FUNCTION_BLOCK TestMotion
VAR_IN_OUT
	axis  : ARRAY [XP .. XM] OF AxisGroup;
	nextInstruct, abortRequest, resetRequest, startRequest, stopRequest: BOOL;
	homeRequest : BYTE;
		
	//statemachine
	stateLVL1 : INT;
	
END_VAR
VAR_INPUT

	speed : LREAL;	

END_VAR
VAR_OUTPUT
END_VAR
VAR
	 //used in tracking Action
	 xorResult : BOOL;
	
	//state-machine
	stateLVL2 : INT;
	initStateLVL2 : BOOL;
	motionBusy : BOOL;
	
	//counter
	i 	: INT :=0;
	
	//used in homeShutter Action
	homeDelay : TON;

END_VAR
VAR CONSTANT
	BRAKE_OFF_C		: BOOL	:= TRUE;
	BRAKE_ON_C		: BOOL	:= FALSE;
	SCAN_VEL_C		: LREAL := 60;
	HOME_VEL_C		: LREAL	:= 3;
	CALIBRATE_VEL_C	: LREAL	:= 100;
	POSITION_VEL_C	: LREAL := 300;
	POS_START_C		: LREAL := 0;
	POS_END_C		: LREAL := 751;
	HOMEOFFSET_XP_C	: LREAL	:= (POS_START_C+35);
	HOMEOFFSET_XM_C	: LREAL	:= (POS_END_C-84);
	
	//SIZE_HALL_SW_C 	: LREAL := SIZEOF(GVL.hallPosCalXP);
	
	//For indexing axis
	XP : INT := 0;
	XM : INT := 1;
END_VAR

(*
This function block contains all the motion of the shutter. There are two state machine in this module - stateLVL1 and stateLVL2.
stateLVL1 is used to switch between motions. stateLVL2 is used to operate the statemachine within the particular motion.
Motions are split into different action objects for readibility and maintainability. 
*)

//update Axis_Ref status
axis[XP].axisRef.ReadStatus();
axis[XM].axisRef.ReadStatus();

//reset input
IF abortRequest THEN
	abortRequest := FALSE;
	stateLVL1 := -1; 
END_IF
IF resetRequest THEN
	resetRequest := FALSE;
	stateLVL1 := 0;
END_IF

(*Case statement for motions. There are two level of state. LVL1 located here and LVL2 which are in the ACTION files.*)
CASE stateLVL1 OF
	-1: //Abort state. Disable movement
		axis[XP].mcPower(Axis := axis[XP].axisRef, Enable := TRUE, Enable_Positive := FALSE, Enable_Negative := FALSE);
		axis[XM].mcPower(Axis := axis[XM].axisRef, Enable := TRUE, Enable_Positive := FALSE, Enable_Negative := FALSE);	
		axis[XP].mcHome(Axis := axis[XP].axisRef, Execute := FALSE);
		axis[XM].mcHome(Axis := axis[XP].axisRef, Execute := FALSE);
		axis[XP].mcReset(Axis := axis[XP].axisRef, Execute := FALSE);
		axis[XM].mcReset(Axis := axis[XM].axisRef, Execute := FALSE);
		axis[XP].brake 	:= BRAKE_ON_C;
		axis[XM].brake 	:= BRAKE_ON_C;
		nextInstruct 	:= FALSE;
		GVL.fbWaitTimer(IN:=FALSE);
		
	0: //reset state
		motionBusy := FALSE;
		initStateLVL2 := FALSE;
		nextInstruct := FALSE;
		axis[XP].mcReset(Axis := axis[XP].axisRef, Execute := TRUE, ErrorID => axis[XP].errorID);
		axis[XM].mcReset(Axis := axis[XM].axisRef, Execute := TRUE, ErrorID => axis[XM].errorID);
		IF axis[XP].mcReset.Error OR axis[XM].mcReset.Error THEN
			axis[XP].mcPower(Axis := axis[XP].axisRef, Enable := TRUE, Enable_Positive := FALSE, Enable_Negative := FALSE);
			axis[XM].mcPower(Axis := axis[XM].axisRef, Enable := TRUE, Enable_Positive := FALSE, Enable_Negative := FALSE);
			axis[XP].brake 	:= BRAKE_ON_C;
			axis[XM].brake 	:= BRAKE_ON_C;
			stateLVL1 		:= -1; //go to stop state
			stateLVL2		:=0;

			//Should report an error flag go to error handle state
		ELSIF axis[XP].mcReset.Done AND axis[XM].mcReset.Done THEN
			axis[XP].mcPower(Axis := axis[XP].axisRef, Enable := TRUE, Enable_Positive := TRUE, Enable_Negative := TRUE);
			axis[XM].mcPower(Axis := axis[XM].axisRef, Enable := TRUE, Enable_Positive := TRUE, Enable_Negative := TRUE);
			axis[XP].mcReset(Axis := axis[XP].axisRef, Execute := FALSE);
			axis[XM].mcReset(Axis := axis[XM].axisRef, Execute := FALSE);
			axis[XP].brake := BRAKE_OFF_C;
			axis[XM].brake := BRAKE_OFF_C;
			axis[XP].mcStop(Axis:=axis[XP].axisRef, Execute:=FALSE);
			axis[XM].mcStop(Axis:=axis[XM].axisRef, Execute:=FALSE);
			stateLVL1 	:= 100; //go to stop state
			stateLVL2	:=0;		
			GVL.fbWaitTimer(IN:=FALSE);	
		END_IF
		
	100: //stop state
		axis[XP].mcMoveAbs(Axis := axis[XP].axisRef, Execute := FALSE);
		axis[XM].mcMoveAbs(Axis := axis[XM].axisRef, Execute := FALSE);
		axis[XP].mcJog(Axis:=axis[XP].axisRef, JogForward:=FALSE, JogBackwards:=FALSE);
		axis[XM].mcJog(Axis:=axis[XM].axisRef, JogForward:=FALSE, JogBackwards:=FALSE);
		axis[XP].mcHome(Axis := axis[XP].axisRef, Execute := FALSE);
		axis[XM].mcHome(Axis := axis[XP].axisRef, Execute := FALSE);
		stateLVL2 := 0;
		GVL.fbWaitTimer(IN:=FALSE);
	
	400: //Homing start for both blades
		homeShutter();
		IF motionBusy = FALSE THEN
			stateLVL1:=100;
		END_IF


	//States higher than 400 requires HOMING ROUTINE to be ran first.
	//////////////////////////////////////////////////////////////////////////////////////////////
	//Basic Motions
	//////////////////////////////////////////////////////////////////////////////////////////////	

	1000: //Open shutter
		openShutter();
		IF motionBusy = FALSE THEN
			stateLVL1:=100;
		END_IF
		
	1100: //Close shutter towards X+ side. 
		closeShutterPlus();
		IF motionBusy = FALSE THEN
			stateLVL1:=100;
		END_IF
		
	1200: //Close shutter towards X- side. 
		closeShutterMinus();
		IF motionBusy = FALSE THEN
			stateLVL1:=100;
		END_IF
		
	1300: //AxisXP absolute move
		axis[XP].mcMoveAbs(Axis:=axis[XP].axisRef, Position:=GVL.setPosition, Velocity:=speed, Execute:=TRUE);
		IF axis[XP].mcMoveAbs.Done THEN
			axis[XP].mcMoveAbs(Axis:=axis[XP].axisRef, Execute:=FALSE);
			stateLVL1 := 100;
		END_IF

	1400: //AxisXM move absolute
		axis[XM].mcMoveAbs(Axis:=axis[XM].axisRef, Position:=GVL.setPosition, Velocity:=speed, Execute:=TRUE);
		IF axis[XM].mcMoveAbs.Done THEN
			axis[XM].mcMoveAbs(Axis:=axis[XM].axisRef, Execute:=FALSE);
			stateLVL1 := 100;
		END_IF

	1500: //AxisXP Jog Forward
		axis[XP].mcJog(Axis:=axis[XP].axisRef, JogForward:=TRUE, JogBackwards:=FALSE, Mode:=MC_JOGMODE_STANDARD_SLOW);
	
	1600: //AxisXP Jog Backward
		axis[XP].mcJog(Axis:=axis[XP].axisRef, JogForward:=FALSE, JogBackwards:=TRUE, Mode:=MC_JOGMODE_STANDARD_SLOW);
		
	1700: //AxisXM Jog Backward
		axis[XM].mcJog(Axis:=axis[XM].axisRef, JogForward:=TRUE, JogBackwards:=FALSE, Mode:=MC_JOGMODE_STANDARD_SLOW);
	
	1800: //AxisXM Jog Forward
		axis[XM].mcJog(Axis:=axis[XM].axisRef, JogForward:=FALSE, JogBackwards:=TRUE, Mode:=MC_JOGMODE_STANDARD_SLOW);

	
	//////////////////////////////////////////////////////////////////////////////////////////////
	//Motion for visit - NORMAL MODE
	//////////////////////////////////////////////////////////////////////////////////////////////	

	2000:
		visit();
		IF motionBusy = FALSE THEN
			stateLVL1:=100;
		END_IF
	
	//////////////////////////////////////////////////////////////////////////////////////////////
	//Cycler -- for use in testing shutter cycle
	//////////////////////////////////////////////////////////////////////////////////////////////
		
	3100: //Cycler sequence 
		cycler();
		IF motionBusy = FALSE THEN
			stateLVL1:=100;
		END_IF	

	//////////////////////////////////////////////////////////////////////////////////////////////
	//Soft Calibration
	//////////////////////////////////////////////////////////////////////////////////////////////

	8000: //Perform soft calibration
		calibrateXP();
		calibrateXM();
		//openShutter();
		IF motionBusy = FALSE THEN
			stateLVL1:=100;
		END_IF

END_CASE

//track motion of both blades
tracking();

ACTION calibrateXM:
//////////////////////////////////////////////////
//perform software calibration of axisXM blade. //
//////////////////////////////////////////////////

IF initStateLVL2 = FALSE THEN
	initStateLVL2 := TRUE;
	stateLVL2 :=9010;
	motionBusy := TRUE;
END_IF	

CASE stateLVL2 OF
	
	9010: //Clear previous Calibration value
		FOR i:=0 TO GVL.tripCount_C BY 1 DO
			axis[XM].hallPosCal[0,i]:=0;
			axis[XM].hallPosCal[1,i]:=0;
		END_FOR
		axis[XM].tripCount := 0;
		axis[XM].isCalibrated := FALSE;
		stateLVL2:=9020;
		
	9020: //Put Shutter in Open Position
		axis[XP].mcMoveAbs(Axis:=axis[XP].axisRef, Position:= POS_START_C, Velocity:=POSITION_VEL_C, Execute:=TRUE);
		axis[XM].mcMoveAbs(Axis:=axis[XM].axisRef, Position:= POS_END_C, Velocity:=POSITION_VEL_C, Execute:=TRUE);
		IF axis[XP].mcMoveAbs.Done AND axis[XM].mcMoveAbs.Done THEN
			axis[XP].mcMoveAbs(Axis:=axis[XP].axisRef, Execute:=FALSE);
			axis[XM].mcMoveAbs(Axis:=axis[XM].axisRef, Execute:=FALSE);
			stateLVL2:=9030;
		END_IF
		
		//This section is required to get rid of false trigger when system starts up
		FOR i:=GVL.hallLower_C TO GVL.hallUpper_C BY 1 DO
			axis[XM].hallSigCal_rtrig[i](CLK:=GVL.hallSwitch[i]);
			axis[XM].hallSigCal_ftrig[i](CLK:=GVL.hallSwitch[i]);
			IF axis[XM].hallSigCal_rtrig[i].Q OR axis[XM].hallSigCal_ftrig[i].Q THEN
				; //do nothing
			END_IF
		END_FOR	
	
	9030: //Calibrate AxisXM twoards X+ side.
		//record position and sequence of hall trips at rising and falling edge.
		FOR i:=GVL.hallLower_C TO GVL.hallUpper_C BY 1 DO
			axis[XM].hallSigCal_rtrig[i](CLK:=GVL.hallSwitch[i]);
			axis[XM].hallSigCal_ftrig[i](CLK:=GVL.hallSwitch[i]);
			IF axis[XM].hallSigCal_rtrig[i].Q OR axis[XM].hallSigCal_ftrig[i].Q THEN	
				
				axis[XM].hallSequence[GVL.dirNeg_C, axis[XM].tripCount].0 := axis[XM].hallSigCal_rtrig[0].Q OR axis[XM].hallSigCal_ftrig[0].Q;
				axis[XM].hallSequence[GVL.dirNeg_C, axis[XM].tripCount].1 := axis[XM].hallSigCal_rtrig[1].Q OR axis[XM].hallSigCal_ftrig[1].Q;
				axis[XM].hallSequence[GVL.dirNeg_C, axis[XM].tripCount].2 := axis[XM].hallSigCal_rtrig[2].Q OR axis[XM].hallSigCal_ftrig[2].Q;
				axis[XM].hallSequence[GVL.dirNeg_C, axis[XM].tripCount].3 := axis[XM].hallSigCal_rtrig[3].Q OR axis[XM].hallSigCal_ftrig[3].Q;
				axis[XM].hallSequence[GVL.dirNeg_C, axis[XM].tripCount].4 := axis[XM].hallSigCal_rtrig[4].Q OR axis[XM].hallSigCal_ftrig[4].Q;
				axis[XM].hallSequence[GVL.dirNeg_C, axis[XM].tripCount].5 := axis[XM].hallSigCal_rtrig[5].Q OR axis[XM].hallSigCal_ftrig[5].Q;
				axis[XM].hallSequence[GVL.dirNeg_C, axis[XM].tripCount].6 := axis[XM].hallSigCal_rtrig[6].Q OR axis[XM].hallSigCal_ftrig[6].Q;
				axis[XM].hallSequence[GVL.dirNeg_C, axis[XM].tripCount].7 := axis[XM].hallSigCal_rtrig[7].Q OR axis[XM].hallSigCal_ftrig[7].Q;
				axis[XM].hallSequence[GVL.dirNeg_C, axis[XM].tripCount].8 := axis[XM].hallSigCal_rtrig[8].Q OR axis[XM].hallSigCal_ftrig[8].Q;
				axis[XM].hallSequence[GVL.dirNeg_C, axis[XM].tripCount].9 := axis[XM].hallSigCal_rtrig[9].Q OR axis[XM].hallSigCal_ftrig[9].Q;
				axis[XM].hallSequence[GVL.dirNeg_C, axis[XM].tripCount].10 := axis[XM].hallSigCal_rtrig[10].Q OR axis[XM].hallSigCal_ftrig[10].Q;
				axis[XM].hallSequence[GVL.dirNeg_C, axis[XM].tripCount].11 := axis[XM].hallSigCal_rtrig[11].Q OR axis[XM].hallSigCal_ftrig[11].Q;
				axis[XM].hallSequence[GVL.dirNeg_C, axis[XM].tripCount].12 := axis[XM].hallSigCal_rtrig[12].Q OR axis[XM].hallSigCal_ftrig[12].Q;
				axis[XM].hallSequence[GVL.dirNeg_C, axis[XM].tripCount].13 := axis[XM].hallSigCal_rtrig[13].Q OR axis[XM].hallSigCal_ftrig[13].Q;
				axis[XM].hallSequence[GVL.dirNeg_C, axis[XM].tripCount].14 := axis[XM].hallSigCal_rtrig[14].Q OR axis[XM].hallSigCal_ftrig[14].Q;
				
				axis[XM].hallPosCal[GVL.dirNeg_C, axis[XM].tripCount] := axis[XM].axisRef.NcToPlc.ActPos;
				
				axis[XM].tripCount := axis[XM].tripCount + 1;		

			END_IF
		END_FOR

		//start moving axisXP towards x+ side
		axis[XM].mcMoveAbs(Axis:=axis[XM].axisRef, Position:=POS_START_C, Velocity:=CALIBRATE_VEL_C, Execute:=TRUE);
		IF axis[XM].mcMoveAbs.Done THEN
			axis[XM].mcMoveAbs(Axis:=axis[XP].axisRef, Execute:=FALSE);
			stateLVL2:= 9040;
		END_IF
	
	
	9040: //Calibrate AxisXM twoards X- side.
		//record position and sequence of hall trips at rising and falling edge.
		FOR i:=GVL.hallLower_C TO GVL.hallUpper_C BY 1 DO
			axis[XM].hallSigCal_rtrig[i](CLK:=GVL.hallSwitch[i]);
			axis[XM].hallSigCal_ftrig[i](CLK:=GVL.hallSwitch[i]);
			IF axis[XM].hallSigCal_rtrig[i].Q OR axis[XM].hallSigCal_ftrig[i].Q THEN	
				
				axis[XM].hallSequence[GVL.dirPos_C, axis[XM].tripCount].0 := axis[XM].hallSigCal_rtrig[0].Q OR axis[XM].hallSigCal_ftrig[0].Q;
				axis[XM].hallSequence[GVL.dirPos_C, axis[XM].tripCount].1 := axis[XM].hallSigCal_rtrig[1].Q OR axis[XM].hallSigCal_ftrig[1].Q;
				axis[XM].hallSequence[GVL.dirPos_C, axis[XM].tripCount].2 := axis[XM].hallSigCal_rtrig[2].Q OR axis[XM].hallSigCal_ftrig[2].Q;
				axis[XM].hallSequence[GVL.dirPos_C, axis[XM].tripCount].3 := axis[XM].hallSigCal_rtrig[3].Q OR axis[XM].hallSigCal_ftrig[3].Q;
				axis[XM].hallSequence[GVL.dirPos_C, axis[XM].tripCount].4 := axis[XM].hallSigCal_rtrig[4].Q OR axis[XM].hallSigCal_ftrig[4].Q;
				axis[XM].hallSequence[GVL.dirPos_C, axis[XM].tripCount].5 := axis[XM].hallSigCal_rtrig[5].Q OR axis[XM].hallSigCal_ftrig[5].Q;
				axis[XM].hallSequence[GVL.dirPos_C, axis[XM].tripCount].6 := axis[XM].hallSigCal_rtrig[6].Q OR axis[XM].hallSigCal_ftrig[6].Q;
				axis[XM].hallSequence[GVL.dirPos_C, axis[XM].tripCount].7 := axis[XM].hallSigCal_rtrig[7].Q OR axis[XM].hallSigCal_ftrig[7].Q;
				axis[XM].hallSequence[GVL.dirPos_C, axis[XM].tripCount].8 := axis[XM].hallSigCal_rtrig[8].Q OR axis[XM].hallSigCal_ftrig[8].Q;
				axis[XM].hallSequence[GVL.dirPos_C, axis[XM].tripCount].9 := axis[XM].hallSigCal_rtrig[9].Q OR axis[XM].hallSigCal_ftrig[9].Q;
				axis[XM].hallSequence[GVL.dirPos_C, axis[XM].tripCount].10 := axis[XM].hallSigCal_rtrig[10].Q OR axis[XM].hallSigCal_ftrig[10].Q;
				axis[XM].hallSequence[GVL.dirPos_C, axis[XM].tripCount].11 := axis[XM].hallSigCal_rtrig[11].Q OR axis[XM].hallSigCal_ftrig[11].Q;
				axis[XM].hallSequence[GVL.dirPos_C, axis[XM].tripCount].12 := axis[XM].hallSigCal_rtrig[12].Q OR axis[XM].hallSigCal_ftrig[12].Q;
				axis[XM].hallSequence[GVL.dirPos_C, axis[XM].tripCount].13 := axis[XM].hallSigCal_rtrig[13].Q OR axis[XM].hallSigCal_ftrig[13].Q;
				axis[XM].hallSequence[GVL.dirPos_C, axis[XM].tripCount].14 := axis[XM].hallSigCal_rtrig[14].Q OR axis[XM].hallSigCal_ftrig[14].Q;
			
				axis[XM].hallPosCal[GVL.dirPos_C, axis[XM].tripCount] := axis[XM].axisRef.NcToPlc.ActPos;
				axis[XM].tripCount := axis[XM].tripCount - 1;	
			END_IF
		END_FOR
	
		//start moving axisXP towards x- side
		axis[XM].mcMoveAbs(Axis:=axis[XM].axisRef, Position:=POS_END_C, Velocity:=CALIBRATE_VEL_C, Execute:=TRUE);
		IF axis[XM].mcMoveAbs.Done THEN
			axis[XM].mcMoveAbs(Axis:=axis[XM].axisRef, Execute:=FALSE);
			stateLVL2 := 9050;
		END_IF
		
	9050: 
		axis[XM].mcJog(Axis := axis[XM].axisRef, Mode := MC_JOGMODE_CONTINOUS, Velocity := SCAN_VEL_C, JogBackwards := axis[XM].limitHome);
		IF NOT axis[XM].limitHome THEN
			axis[XM].mcJog(Axis := axis[XM].axisRef, Mode := MC_JOGMODE_CONTINOUS, JogBackwards := FALSE);
			stateLVL2 := 9060;
		END_IF

	9060: //slowly homed back to switch
		axis[XM].mcJog(Axis := axis[XM].axisRef, Mode := MC_JOGMODE_CONTINOUS, Velocity := HOME_VEL_C, JogForward := NOT axis[XM].limitHome);
		IF axis[XM].limitHome THEN
			axis[XM].mcJog(Axis := axis[XM].axisRef, Mode := MC_JOGMODE_CONTINOUS, JogForward := FALSE);
			stateLVL2 := 9070;
			axis[XM].isCalibrated := TRUE;
		END_IF			
		
	9070: //End action
		initStateLVL2 := FALSE;
		stateLVL2 := 0;
		motionBusy := FALSE;


END_CASE
END_ACTION

ACTION calibrateXP:
//////////////////////////////////////////////////
//perform software calibration of axisXP blade. //
//////////////////////////////////////////////////

IF initStateLVL2 = FALSE THEN
	initStateLVL2 := TRUE;
	stateLVL2 :=8010;
	motionBusy := TRUE;
END_IF	

CASE stateLVL2 OF

	8010: //Clear previous Calibration value
		FOR i:=0 TO GVL.tripCount_C BY 1 DO
			axis[XP].hallPosCal[0,i]:=0;
			axis[XP].hallPosCal[1,i]:=0;
		END_FOR
		axis[XP].tripCount := 0;	
		axis[XP].isCalibrated := FALSE;
		stateLVL2:=8020;
		
	8020: //Put Shutter in Open Position
		axis[XP].mcMoveAbs(Axis:=axis[XP].axisRef, Position:= POS_START_C, Velocity:=POSITION_VEL_C, Execute:=TRUE);
		axis[XM].mcMoveAbs(Axis:=axis[XM].axisRef, Position:= POS_END_C, Velocity:=POSITION_VEL_C, Execute:=TRUE);
		IF axis[XP].mcMoveAbs.Done AND axis[XM].mcMoveAbs.Done THEN
			axis[XP].mcMoveAbs(Axis:=axis[XP].axisRef, Execute:=FALSE);
			axis[XM].mcMoveAbs(Axis:=axis[XM].axisRef, Execute:=FALSE);
			stateLVL2:=8030;
		END_IF
		
		//This section is required to get rid of false trigger when system starts up
		FOR i:=GVL.hallLower_C TO GVL.hallUpper_C BY 1 DO
			axis[XP].hallSigCal_rtrig[i](CLK:=GVL.hallSwitch[i]);
			axis[XP].hallSigCal_ftrig[i](CLK:=GVL.hallSwitch[i]);
			IF axis[XP].hallSigCal_rtrig[i].Q OR axis[XP].hallSigCal_ftrig[i].Q THEN
				; //do nothing
			END_IF
		END_FOR

	8030: //Calibrate AxisXP towards X- side.
		//record position and sequence of hall trips at rising and falling edge.
		FOR i:=GVL.hallLower_C TO GVL.hallUpper_C BY 1 DO
			axis[XP].hallSigCal_rtrig[i](CLK:=GVL.hallSwitch[i]);
			axis[XP].hallSigCal_ftrig[i](CLK:=GVL.hallSwitch[i]);
			IF axis[XP].hallSigCal_rtrig[i].Q OR axis[XP].hallSigCal_ftrig[i].Q THEN	

				axis[XP].hallSequence[GVL.dirPos_C, axis[XP].tripCount].0 := axis[XP].hallSigCal_rtrig[0].Q OR axis[XP].hallSigCal_ftrig[0].Q;
				axis[XP].hallSequence[GVL.dirPos_C, axis[XP].tripCount].1 := axis[XP].hallSigCal_rtrig[1].Q OR axis[XP].hallSigCal_ftrig[1].Q;
				axis[XP].hallSequence[GVL.dirPos_C, axis[XP].tripCount].2 := axis[XP].hallSigCal_rtrig[2].Q OR axis[XP].hallSigCal_ftrig[2].Q;
				axis[XP].hallSequence[GVL.dirPos_C, axis[XP].tripCount].3 := axis[XP].hallSigCal_rtrig[3].Q OR axis[XP].hallSigCal_ftrig[3].Q;
				axis[XP].hallSequence[GVL.dirPos_C, axis[XP].tripCount].4 := axis[XP].hallSigCal_rtrig[4].Q OR axis[XP].hallSigCal_ftrig[4].Q;
				axis[XP].hallSequence[GVL.dirPos_C, axis[XP].tripCount].5 := axis[XP].hallSigCal_rtrig[5].Q OR axis[XP].hallSigCal_ftrig[5].Q;
				axis[XP].hallSequence[GVL.dirPos_C, axis[XP].tripCount].6 := axis[XP].hallSigCal_rtrig[6].Q OR axis[XP].hallSigCal_ftrig[6].Q;
				axis[XP].hallSequence[GVL.dirPos_C, axis[XP].tripCount].7 := axis[XP].hallSigCal_rtrig[7].Q OR axis[XP].hallSigCal_ftrig[7].Q;
				axis[XP].hallSequence[GVL.dirPos_C, axis[XP].tripCount].8 := axis[XP].hallSigCal_rtrig[8].Q OR axis[XP].hallSigCal_ftrig[8].Q;
				axis[XP].hallSequence[GVL.dirPos_C, axis[XP].tripCount].9 := axis[XP].hallSigCal_rtrig[9].Q OR axis[XP].hallSigCal_ftrig[9].Q;
				axis[XP].hallSequence[GVL.dirPos_C, axis[XP].tripCount].10 := axis[XP].hallSigCal_rtrig[10].Q OR axis[XP].hallSigCal_ftrig[10].Q;
				axis[XP].hallSequence[GVL.dirPos_C, axis[XP].tripCount].11 := axis[XP].hallSigCal_rtrig[11].Q OR axis[XP].hallSigCal_ftrig[11].Q;
				axis[XP].hallSequence[GVL.dirPos_C, axis[XP].tripCount].12 := axis[XP].hallSigCal_rtrig[12].Q OR axis[XP].hallSigCal_ftrig[12].Q;
				axis[XP].hallSequence[GVL.dirPos_C, axis[XP].tripCount].13 := axis[XP].hallSigCal_rtrig[13].Q OR axis[XP].hallSigCal_ftrig[13].Q;
				axis[XP].hallSequence[GVL.dirPos_C, axis[XP].tripCount].14 := axis[XP].hallSigCal_rtrig[14].Q OR axis[XP].hallSigCal_ftrig[14].Q;

				axis[XP].hallPosCal[GVL.dirPos_C, axis[XP].tripCount] := axis[XP].axisRef.NcToPlc.ActPos;
				axis[XP].tripCount := axis[XP].tripCount + 1;		

			END_IF
		END_FOR
	
		//start moving axisXP towards x- side
		axis[XP].mcMoveAbs(Axis:=axis[XP].axisRef, Position:=POS_END_C, Velocity:=CALIBRATE_VEL_C, Execute:=TRUE);
		IF axis[XP].mcMoveAbs.Done THEN
			axis[XP].mcMoveAbs(Axis:=axis[XP].axisRef, Execute:=FALSE);
			stateLVL2:= 8040;
		END_IF
	
	8040: //Calibrate AxisXP towards X+ side.
		//record position and sequence of hall trips at rising and falling edge
		FOR i:=GVL.hallLower_C TO GVL.hallUpper_C BY 1 DO
			axis[XP].hallSigCal_rtrig[i](CLK:=GVL.hallSwitch[i]);
			axis[XP].hallSigCal_ftrig[i](CLK:=GVL.hallSwitch[i]);
			IF axis[XP].hallSigCal_rtrig[i].Q OR axis[XP].hallSigCal_ftrig[i].Q THEN
				
				axis[XP].hallSequence[GVL.dirNeg_C, axis[XP].tripCount].0 := axis[XP].hallSigCal_rtrig[0].Q OR axis[XP].hallSigCal_ftrig[0].Q;
				axis[XP].hallSequence[GVL.dirNeg_C, axis[XP].tripCount].1 := axis[XP].hallSigCal_rtrig[1].Q OR axis[XP].hallSigCal_ftrig[1].Q;
				axis[XP].hallSequence[GVL.dirNeg_C, axis[XP].tripCount].2 := axis[XP].hallSigCal_rtrig[2].Q OR axis[XP].hallSigCal_ftrig[2].Q;
				axis[XP].hallSequence[GVL.dirNeg_C, axis[XP].tripCount].3 := axis[XP].hallSigCal_rtrig[3].Q OR axis[XP].hallSigCal_ftrig[3].Q;
				axis[XP].hallSequence[GVL.dirNeg_C, axis[XP].tripCount].4 := axis[XP].hallSigCal_rtrig[4].Q OR axis[XP].hallSigCal_ftrig[4].Q;
				axis[XP].hallSequence[GVL.dirNeg_C, axis[XP].tripCount].5 := axis[XP].hallSigCal_rtrig[5].Q OR axis[XP].hallSigCal_ftrig[5].Q;
				axis[XP].hallSequence[GVL.dirNeg_C, axis[XP].tripCount].6 := axis[XP].hallSigCal_rtrig[6].Q OR axis[XP].hallSigCal_ftrig[6].Q;
				axis[XP].hallSequence[GVL.dirNeg_C, axis[XP].tripCount].7 := axis[XP].hallSigCal_rtrig[7].Q OR axis[XP].hallSigCal_ftrig[7].Q;
				axis[XP].hallSequence[GVL.dirNeg_C, axis[XP].tripCount].8 := axis[XP].hallSigCal_rtrig[8].Q OR axis[XP].hallSigCal_ftrig[8].Q;
				axis[XP].hallSequence[GVL.dirNeg_C, axis[XP].tripCount].9 := axis[XP].hallSigCal_rtrig[9].Q OR axis[XP].hallSigCal_ftrig[9].Q;
				axis[XP].hallSequence[GVL.dirNeg_C, axis[XP].tripCount].10 := axis[XP].hallSigCal_rtrig[10].Q OR axis[XP].hallSigCal_ftrig[10].Q;
				axis[XP].hallSequence[GVL.dirNeg_C, axis[XP].tripCount].11 := axis[XP].hallSigCal_rtrig[11].Q OR axis[XP].hallSigCal_ftrig[11].Q;
				axis[XP].hallSequence[GVL.dirNeg_C, axis[XP].tripCount].12 := axis[XP].hallSigCal_rtrig[12].Q OR axis[XP].hallSigCal_ftrig[12].Q;
				axis[XP].hallSequence[GVL.dirNeg_C, axis[XP].tripCount].13 := axis[XP].hallSigCal_rtrig[13].Q OR axis[XP].hallSigCal_ftrig[13].Q;
				axis[XP].hallSequence[GVL.dirNeg_C, axis[XP].tripCount].14 := axis[XP].hallSigCal_rtrig[14].Q OR axis[XP].hallSigCal_ftrig[14].Q;
			
				axis[XP].hallPosCal[GVL.dirNeg_C, axis[XP].tripCount] := axis[XP].axisRef.NcToPlc.ActPos;
				axis[XP].tripCount := axis[XP].tripCount - 1;	
			END_IF
		END_FOR
	
		//start moving axisXP towards x+ side
		axis[XP].mcMoveAbs(Axis:=axis[XP].axisRef, Position:=POS_START_C, Velocity:=CALIBRATE_VEL_C, Execute:=TRUE);
		IF axis[XP].mcMoveAbs.Done THEN
			axis[XP].mcMoveAbs(Axis:=axis[XP].axisRef, Execute:=FALSE);
			stateLVL2 := 8050;
		END_IF
	
	8050: 
		axis[XP].mcJog(Axis := axis[XP].axisRef, Mode := MC_JOGMODE_CONTINOUS, Velocity := SCAN_VEL_C, JogForward := axis[XP].limitHome);
		IF NOT axis[XP].limitHome THEN
			axis[XP].mcJog(Axis := axis[XM].axisRef, Mode := MC_JOGMODE_CONTINOUS, JogForward := FALSE);
			stateLVL2 := 8060;
		END_IF

	8060: //slowly homed back to switch
		axis[XP].mcJog(Axis := axis[XP].axisRef, Mode := MC_JOGMODE_CONTINOUS, Velocity := HOME_VEL_C, JogBackwards := NOT axis[XP].limitHome);
		IF axis[XP].limitHome THEN
			axis[XP].mcJog(Axis := axis[XP].axisRef, Mode := MC_JOGMODE_CONTINOUS, JogBackwards := FALSE);
			stateLVL2 := 8070;
			axis[XP].isCalibrated := TRUE;
		END_IF			
		
	8070: //End action
		initStateLVL2 := FALSE;
		stateLVL2 := 0;
		motionBusy := FALSE;

	
END_CASE
END_ACTION

ACTION closeShutterMinus:
//////////////////////////////////////////////////
//Closes shutter in -X position					//
//////////////////////////////////////////////////

IF initStateLVL2 = FALSE THEN
	initStateLVL2 := TRUE;
	stateLVL2 :=1210;
	motionBusy := TRUE;
END_IF

CASE stateLVL2 OF
	
	1210://Close shutter towards X- side. AxisXM retracts to its HOME position (~750 mm)
		axis[XM].mcMoveAbs(Axis:=axis[XM].axisRef, Position:= POS_END_C, Velocity:=speed, Execute:=TRUE);
		IF axis[XM].mcMoveAbs.Done THEN
			axis[XM].mcMoveAbs(Axis:=axis[XM].axisRef, Execute:=FALSE);
			stateLVL2:=1220;
		END_IF
		
	1220: //Close shutter towards X- side. AxisXP extends to its DEPLOYED position
		axis[XP].mcMoveAbs(Axis:=axis[XP].axisRef, Position:= POS_END_C, Velocity:=speed, Execute:=TRUE);
		IF axis[XP].mcMoveAbs.Done THEN
			axis[XP].mcMoveAbs(Axis:=axis[XP].axisRef, Execute:=FALSE);
			stateLVL2 := 1230;
		END_IF
		
	1230: //End Action
		initStateLVL2 := FALSE;
		stateLVL2 := 0;
		motionBusy := FALSE;
END_CASE
END_ACTION

ACTION closeShutterPlus:
//////////////////////////////////////////////////
//Closes shutter in +X position					//
//////////////////////////////////////////////////

IF initStateLVL2 = FALSE THEN
	initStateLVL2 := TRUE;
	stateLVL2 :=1110;
	motionBusy := TRUE;
END_IF

CASE stateLVL2 OF
	
	1110: //Close shutter towards X+ side. axisXP retracts to its HOME position
		axis[XP].mcMoveAbs(Axis:=axis[XP].axisRef, Position:= POS_START_C, Velocity:=speed, Execute:=TRUE);
		IF axis[XP].mcMoveAbs.Done THEN
			axis[XP].mcMoveAbs(Axis:=axis[XP].axisRef, Execute:=FALSE);
			stateLVL2:=1120;
		END_IF
		
	1120: //Close shutter towards X+ side. AxisXM extends to its DEPLOYED position 
		axis[XM].mcMoveAbs(Axis:=axis[XM].axisRef, Position:= POS_START_C, Velocity:=speed, Execute:=TRUE);
		IF axis[XM].mcMoveAbs.Done THEN
			axis[XM].mcMoveAbs(Axis:=axis[XM].axisRef, Execute:=FALSE);
			stateLVL2 := 1130;
		END_IF
	
	1130: //End Action
		initStateLVL2 := FALSE;
		stateLVL2 := 0;
		motionBusy := FALSE;
END_CASE
END_ACTION

ACTION cycler:
///////////////////////////////////////////////////////
//Performs open/close motion until commanded to stop.//
///////////////////////////////////////////////////////

IF initStateLVL2 = FALSE THEN
	initStateLVL2 := TRUE;
	stateLVL2 :=3010;
	motionBusy := TRUE;
END_IF	

CASE stateLVL2 OF

	3010: 
		motionBusy := TRUE;
		GVL.fbWaitTimer(IN:=TRUE, PT:=GVL.expoTime,);
		axis[XM].mcMoveAbs(Axis:=axis[XM].axisRef, Position:= POS_END_C, Velocity:=speed, Execute:=TRUE);
		IF GVL.fbWaitTimer.Q THEN
			axis[XP].mcMoveAbs(Axis:=axis[XP].axisRef, Position:= POS_END_C, Velocity:=speed, Execute:=TRUE);
		END_IF
		IF axis[XP].mcMoveAbs.Done AND axis[XM].mcMoveAbs.Done THEN
			GVL.strokeXP := GVL.strokeXP + 1;
			GVL.strokeXM := GVL.strokeXM + 1;
			GVL.fbWaitTimer(IN:=FALSE);
			axis[XP].mcMoveAbs(Axis:=axis[XP].axisRef, Execute:=FALSE);
			axis[XM].mcMoveAbs(Axis:=axis[XM].axisRef, Execute:=FALSE);
			stateLVL2:=3020;
		END_IF
		
	3020:
		GVL.fbWaitTimer(IN:=TRUE, PT:=T#100MS,);
		IF GVL.fbWaitTimer.Q THEN
			GVL.fbWaitTimer(IN:=FALSE);
			IF stopRequest THEN
				stopRequest:=FALSE;
				stateLVL2:=3999;
			ELSE
				stateLVL2:=3030;
			END_IF
		END_IF
		
	3030: 
		GVL.fbWaitTimer(IN:=TRUE, PT:=GVL.expoTime,);
		axis[XP].mcMoveAbs(Axis:=axis[XP].axisRef, Position:= POS_START_C, Velocity:=speed, Execute:=TRUE);
		IF GVL.fbWaitTimer.Q THEN
			axis[XM].mcMoveAbs(Axis:=axis[XM].axisRef, Position:= POS_START_C, Velocity:=speed, Execute:=TRUE);
		END_IF
		IF axis[XP].mcMoveAbs.Done AND axis[XM].mcMoveAbs.Done THEN
			GVL.strokeXP := GVL.strokeXP + 1;
			GVL.strokeXM := GVL.strokeXM + 1;
			GVL.fbWaitTimer(IN:=FALSE);
			axis[XP].mcMoveAbs(Axis:=axis[XP].axisRef, Execute:=FALSE);
			axis[XM].mcMoveAbs(Axis:=axis[XM].axisRef, Execute:=FALSE);
			stateLVL2:=3040;
		END_IF	
		
	3040:
		GVL.fbWaitTimer(IN:=TRUE, PT:=T#100MS,);
		IF GVL.fbWaitTimer.Q THEN
			GVL.fbWaitTimer(IN:=FALSE);
			IF stopRequest THEN
				stopRequest:=FALSE;
				stateLVL2:=3999;
			ELSE
				stateLVL2:=3010;
			END_IF
		END_IF

		
	3999: //End action
		initStateLVL2 := FALSE;
		stateLVL2 := 0;
		motionBusy := FALSE;
END_CASE
END_ACTION

ACTION homeShutter:
//////////////////////////////////////////////////
//Performs homing routine						//
//////////////////////////////////////////////////

IF initStateLVL2 = FALSE THEN
	initStateLVL2 := TRUE;
	stateLVL2 :=410;
	motionBusy := TRUE;
END_IF	

CASE stateLVL2 OF
	
	410: //Clear Homed flag and calibrated flag
		axis[XP].mcHome(Axis := axis[XP].axisRef, HomingMode := MC_ResetCalibration, bCalibrationCam := TRUE, Execute := TRUE);
		axis[XM].mcHome(Axis := axis[XM].axisRef, HomingMode := MC_ResetCalibration, bCalibrationCam := TRUE, Execute := TRUE);
		axis[XP].isCalibrated := FALSE;
		axis[XM].isCalibrated := FALSE;
		IF axis[XP].mcHome.Done AND axis[XM].mcHome.Done THEN
			stateLVL2 := 420;
		END_IF
		
	420: //Scan for home switch
		axis[XP].mcHome(Axis := axis[XP].axisRef, Execute := FALSE);
		axis[XM].mcHome(Axis := axis[XM].axisRef, Execute := FALSE);
		axis[XP].mcJog(Axis := axis[XP].axisRef, Mode := MC_JOGMODE_CONTINOUS, Velocity := SCAN_VEL_C, JogBackwards := NOT axis[XP].limitHome);
		axis[XM].mcJog(Axis := axis[XM].axisRef, Mode := MC_JOGMODE_CONTINOUS, Velocity := SCAN_VEL_C, JogForward := NOT axis[XM].limitHome);
		IF axis[XP].limitHome AND axis[XM].limitHome THEN
			axis[XP].mcJog(Axis := axis[XP].axisRef, Mode := MC_JOGMODE_CONTINOUS, JogBackwards := FALSE);
			axis[XM].mcJog(Axis := axis[XM].axisRef, Mode := MC_JOGMODE_CONTINOUS, JogForward := FALSE);
			stateLVL2 := 430;
		END_IF

	430: //back off from switch
		axis[XP].mcJog(Axis := axis[XP].axisRef, Mode := MC_JOGMODE_CONTINOUS, Velocity := SCAN_VEL_C, JogForward := axis[XP].limitHome);
		axis[XM].mcJog(Axis := axis[XM].axisRef, Mode := MC_JOGMODE_CONTINOUS, Velocity := SCAN_VEL_C, JogBackwards := axis[XM].limitHome);
		IF NOT axis[XP].limitHome AND NOT axis[XM].limitHome THEN
			axis[XP].mcJog(Axis := axis[XP].axisRef, Mode := MC_JOGMODE_CONTINOUS, JogForward := FALSE);
			axis[XM].mcJog(Axis := axis[XM].axisRef, Mode := MC_JOGMODE_CONTINOUS, JogBackwards := FALSE);
			stateLVL2 := 440;
		END_IF
		
	440: //slowly homed back to switch
		axis[XP].mcJog(Axis := axis[XP].axisRef, Mode := MC_JOGMODE_CONTINOUS, Velocity := HOME_VEL_C, JogBackwards := NOT axis[XP].limitHome);
		axis[XM].mcJog(Axis := axis[XM].axisRef, Mode := MC_JOGMODE_CONTINOUS, Velocity := HOME_VEL_C, JogForward := NOT axis[XM].limitHome);
		IF axis[XP].limitHome AND axis[XM].limitHome THEN
			axis[XP].mcJog(Axis := axis[XP].axisRef, Mode := MC_JOGMODE_CONTINOUS, JogBackwards := FALSE);
			axis[XM].mcJog(Axis := axis[XM].axisRef, Mode := MC_JOGMODE_CONTINOUS, JogForward := FALSE);
			stateLVL2 := 450;
		END_IF	

	450://delay
		homeDelay(IN:=TRUE, PT:=T#100MS);
		IF homeDelay.Q THEN
			homeDelay(IN:=FALSE);	
			stateLVL2 := 460;
		END_IF
		
	460://set home
		axis[XP].mcHome(Axis := axis[XP].axisRef, Position := POS_START_C, HomingMode := MC_DIRECT, Execute := TRUE);
		axis[XM].mcHome(Axis := axis[XM].axisRef, Position := POS_END_C, HomingMode := MC_DIRECT, Execute := TRUE);	
		IF axis[XP].mcHome.Done AND axis[XM].mcHome.Done THEN
			axis[XP].mcHome(Axis := axis[XP].axisRef, Execute := FALSE);
			axis[XM].mcHome(Axis := axis[XM].axisRef, Execute := FALSE);
			stateLVL2 := 470;
		END_IF	
		
		
	470: //End Action
		initStateLVL2 := FALSE;
		stateLVL2 := 0;
		motionBusy := FALSE;
END_CASE
END_ACTION

ACTION openShutter:
//////////////////////////////////////////////////
//Puts shutter in open position					//
//////////////////////////////////////////////////

IF initStateLVL2 = FALSE THEN
	initStateLVL2 := TRUE;
	stateLVL2 :=1010;
	motionBusy := TRUE;
END_IF	

CASE stateLVL2 OF
	
	1010:
		motionBusy := TRUE;
		axis[XP].mcMoveAbs(Axis:=axis[XP].axisRef, Position:= POS_START_C, Velocity:=speed, Execute:=TRUE);
		axis[XM].mcMoveAbs(Axis:=axis[XM].axisRef, Position:= POS_END_C, Velocity:=speed, Execute:=TRUE);
		IF axis[XP].mcMoveAbs.Done AND axis[XM].mcMoveAbs.Done THEN
			axis[XP].mcMoveAbs(Axis:=axis[XP].axisRef, Execute:=FALSE);
			axis[XM].mcMoveAbs(Axis:=axis[XM].axisRef, Execute:=FALSE);
			stateLVL2 := 1020;
		END_IF	
		
	1020: //End action
		initStateLVL2 := FALSE;
		stateLVL2 := 0;
		motionBusy := FALSE;
		
END_CASE
END_ACTION

ACTION tracking:
//////////////////////////////////////////////////////////////
//Algorithm for tracking blade position using hall switches	//
//////////////////////////////////////////////////////////////

//Only one hall will ever trip for 1 set of blades. This flag is used to make sure the trip increment only once per cycle.
axis[XP].trackedFlag := FALSE;
axis[XM].trackedFlag := FALSE;

//Hall sensors position tracking for axis XP
FOR i:=GVL.hallLower_C TO GVL.hallUpper_C BY 1 DO
	axis[XP].hallSigCal_rtrig[i](CLK:=GVL.hallSwitch[i]);
	axis[XP].hallSigCal_ftrig[i](CLK:=GVL.hallSwitch[i]);
	IF (axis[XP].hallSigCal_rtrig[i].Q OR axis[XP].hallSigCal_ftrig[i].Q) AND axis[XP].axisRef.Status.Moving THEN
		axis[XP].trackedFlag := TRUE;
	END_IF
END_FOR
	
IF axis[XP].trackedFlag THEN
	//record trigger status of each hall sensor into hallSequence for comparing;
	GVL.hallSequence.0 := axis[XP].hallSigCal_rtrig[0].Q OR axis[XP].hallSigCal_ftrig[0].Q;
	GVL.hallSequence.1 := axis[XP].hallSigCal_rtrig[1].Q OR axis[XP].hallSigCal_ftrig[1].Q;
	GVL.hallSequence.2 := axis[XP].hallSigCal_rtrig[2].Q OR axis[XP].hallSigCal_ftrig[2].Q;
	GVL.hallSequence.3 := axis[XP].hallSigCal_rtrig[3].Q OR axis[XP].hallSigCal_ftrig[3].Q;
	GVL.hallSequence.4 := axis[XP].hallSigCal_rtrig[4].Q OR axis[XP].hallSigCal_ftrig[4].Q;
	GVL.hallSequence.5 := axis[XP].hallSigCal_rtrig[5].Q OR axis[XP].hallSigCal_ftrig[5].Q;
	GVL.hallSequence.6 := axis[XP].hallSigCal_rtrig[6].Q OR axis[XP].hallSigCal_ftrig[6].Q;
	GVL.hallSequence.7 := axis[XP].hallSigCal_rtrig[7].Q OR axis[XP].hallSigCal_ftrig[7].Q;
	GVL.hallSequence.8 := axis[XP].hallSigCal_rtrig[8].Q OR axis[XP].hallSigCal_ftrig[8].Q;
	GVL.hallSequence.9 := axis[XP].hallSigCal_rtrig[9].Q OR axis[XP].hallSigCal_ftrig[9].Q;
	GVL.hallSequence.10 := axis[XP].hallSigCal_rtrig[10].Q OR axis[XP].hallSigCal_ftrig[10].Q;
	GVL.hallSequence.11 := axis[XP].hallSigCal_rtrig[11].Q OR axis[XP].hallSigCal_ftrig[11].Q;
	GVL.hallSequence.12 := axis[XP].hallSigCal_rtrig[12].Q OR axis[XP].hallSigCal_ftrig[12].Q;
	GVL.hallSequence.13 := axis[XP].hallSigCal_rtrig[13].Q OR axis[XP].hallSigCal_ftrig[13].Q;
	GVL.hallSequence.14 := axis[XP].hallSigCal_rtrig[14].Q OR axis[XP].hallSigCal_ftrig[14].Q;	

	(* Unary XOR of hallSequence. With one blade running, 1 bit should be HIGH at a time .
		Result of 1 indicates presence of one blade sequence. Result of 0 indicates presence of two blade sequence *)
	xorResult := (GVL.hallSequence.0 XOR GVL.hallSequence.1 XOR GVL.hallSequence.2 XOR GVL.hallSequence.3 XOR GVL.hallSequence.4 XOR
		GVL.hallSequence.5 XOR GVL.hallSequence.6 XOR GVL.hallSequence.7 XOR GVL.hallSequence.8 XOR GVL.hallSequence.9 XOR
		GVL.hallSequence.10 XOR GVL.hallSequence.11 XOR GVL.hallSequence.12 XOR GVL.hallSequence.13 XOR GVL.hallSequence.14);
	IF xorResult THEN
		axis[XP].seqToCompare := GVL.hallSequence;
	ELSIF axis[XM].axisRef.status.PositiveDirection THEN
		axis[XP].seqToCompare := (GVL.hallSequence XOR axis[XM].hallSequence[GVL.dirPos_C, axis[XM].tripCount]);//+1 required since XM tripCount does not update until further down
	ELSIF axis[XM].axisRef.status.NegativeDirection THEN
		axis[XP].seqToCompare := (GVL.hallSequence XOR axis[XM].hallSequence[GVL.dirNeg_C, axis[XM].tripCount]);	
	ELSE
		; //Should generate error code here
	END_IF	

	//Compare current sequence with recorded sequence. Update position if match.
	IF axis[XP].axisRef.status.PositiveDirection AND axis[XP].hallSequence[GVL.dirPos_C, axis[XP].tripCount] = axis[XP].seqToCompare THEN
		axis[XP].hallPosAct := axis[XP].hallPosCal[GVL.dirPos_C, axis[XP].tripCount];
		axis[XP].tripCount := axis[XP].tripCount + 1;	
		//track difference between hall sensor and encoder data at trip point
		axis[XP].posDiffAtTrip := axis[XP].axisRef.NcToPlc.ActPos - axis[XP].hallPosAct;
	END_IF
	IF axis[XP].axisRef.status.NegativeDirection AND axis[XP].hallSequence[GVL.dirNeg_C, axis[XP].tripCount] = axis[XP].seqToCompare THEN
		axis[XP].hallPosAct := axis[XP].hallPosCal[GVL.dirNeg_C, axis[XP].tripCount];
		axis[XP].tripCount := axis[XP].tripCount - 1;	
		//track difference between hall sensor and encoder data at trip point
		axis[XP].posDiffAtTrip := axis[XP].axisRef.NcToPlc.ActPos - axis[XP].hallPosAct;
	END_IF
END_IF


//Hall sensors position tracking for axis XM
FOR i:=GVL.hallLower_C TO GVL.hallUpper_C BY 1 DO
	axis[XM].hallSigCal_rtrig[i](CLK:=GVL.hallSwitch[i]);
	axis[XM].hallSigCal_ftrig[i](CLK:=GVL.hallSwitch[i]);
	IF (axis[XM].hallSigCal_rtrig[i].Q OR axis[XM].hallSigCal_ftrig[i].Q) AND axis[XM].axisRef.Status.Moving AND NOT axis[XM].trackedFlag THEN
		axis[XM].trackedFlag := TRUE;
	END_IF
END_FOR

IF axis[XM].trackedFlag THEN
	
	//record trigger status of each hall sensor into hallSequence for comparing;
	GVL.hallSequence.0 := axis[XM].hallSigCal_rtrig[0].Q OR axis[XM].hallSigCal_ftrig[0].Q;
	GVL.hallSequence.1 := axis[XM].hallSigCal_rtrig[1].Q OR axis[XM].hallSigCal_ftrig[1].Q;
	GVL.hallSequence.2 := axis[XM].hallSigCal_rtrig[2].Q OR axis[XM].hallSigCal_ftrig[2].Q;
	GVL.hallSequence.3 := axis[XM].hallSigCal_rtrig[3].Q OR axis[XM].hallSigCal_ftrig[3].Q;
	GVL.hallSequence.4 := axis[XM].hallSigCal_rtrig[4].Q OR axis[XM].hallSigCal_ftrig[4].Q;
	GVL.hallSequence.5 := axis[XM].hallSigCal_rtrig[5].Q OR axis[XM].hallSigCal_ftrig[5].Q;
	GVL.hallSequence.6 := axis[XM].hallSigCal_rtrig[6].Q OR axis[XM].hallSigCal_ftrig[6].Q;
	GVL.hallSequence.7 := axis[XM].hallSigCal_rtrig[7].Q OR axis[XM].hallSigCal_ftrig[7].Q;
	GVL.hallSequence.8 := axis[XM].hallSigCal_rtrig[8].Q OR axis[XM].hallSigCal_ftrig[8].Q;
	GVL.hallSequence.9 := axis[XM].hallSigCal_rtrig[9].Q OR axis[XM].hallSigCal_ftrig[9].Q;
	GVL.hallSequence.10 := axis[XM].hallSigCal_rtrig[10].Q OR axis[XM].hallSigCal_ftrig[10].Q;
	GVL.hallSequence.11 := axis[XM].hallSigCal_rtrig[11].Q OR axis[XM].hallSigCal_ftrig[11].Q;
	GVL.hallSequence.12 := axis[XM].hallSigCal_rtrig[12].Q OR axis[XM].hallSigCal_ftrig[12].Q;
	GVL.hallSequence.13 := axis[XM].hallSigCal_rtrig[13].Q OR axis[XM].hallSigCal_ftrig[13].Q;
	GVL.hallSequence.14 := axis[XM].hallSigCal_rtrig[14].Q OR axis[XM].hallSigCal_ftrig[14].Q;			
	
	(* Unary XOR of hallSequence. With one blade running, 1 bit should be HIGH at a time .
		Result of 1 indicates presence of one blade sequence. Result of 0 indicates presence of two blade sequence *)
	xorResult := GVL.hallSequence.0 XOR GVL.hallSequence.1 XOR GVL.hallSequence.2 XOR GVL.hallSequence.3 XOR GVL.hallSequence.4 XOR
		GVL.hallSequence.5 XOR GVL.hallSequence.6 XOR GVL.hallSequence.7 XOR GVL.hallSequence.8 XOR GVL.hallSequence.9 XOR
		GVL.hallSequence.10 XOR GVL.hallSequence.11 XOR GVL.hallSequence.12 XOR GVL.hallSequence.13 XOR GVL.hallSequence.14;
	IF xorResult THEN
		axis[XM].seqToCompare := GVL.hallSequence;
	ELSIF axis[XP].axisRef.status.PositiveDirection THEN
		axis[XM].seqToCompare := (GVL.hallSequence XOR axis[XP].hallSequence[GVL.dirPos_C, axis[XP].tripCount-1]); //requires -1 since XP tripcount has already incremented
	ELSIF axis[XP].axisRef.status.NegativeDirection THEN
		axis[XM].seqToCompare := (GVL.hallSequence XOR axis[XP].hallSequence[GVL.dirNeg_C, axis[XP].tripCount+1]);	
	ELSE
		; //Should generate error code here
	END_IF		

	//Compare current sequence with recorded sequence. Update position if match.	
	IF axis[XM].axisRef.status.PositiveDirection AND axis[XM].hallSequence[GVL.dirPos_C, axis[XM].tripCount] = axis[XM].seqToCompare THEN
		axis[XM].hallPosAct := axis[XM].hallPosCal[GVL.dirPos_C, axis[XM].tripCount];
		axis[XM].tripCount := axis[XM].tripCount - 1;	
		//track difference between hall sensor and encoder data at trip point
		axis[XM].posDiffAtTrip := axis[XM].axisRef.NcToPlc.ActPos - axis[XM].hallPosAct;
	END_IF
	IF axis[XM].axisRef.status.NegativeDirection AND axis[XM].hallSequence[GVL.dirNeg_C, axis[XM].tripCount] = axis[XM].seqToCompare THEN
		axis[XM].hallPosAct := axis[XM].hallPosCal[GVL.dirNeg_C, axis[XM].tripCount];
		axis[XM].tripCount := axis[XM].tripCount + 1;	
		//track difference between hall sensor and encoder data at trip point
		axis[XM].posDiffAtTrip := axis[XM].axisRef.NcToPlc.ActPos - axis[XM].hallPosAct;
	END_IF
END_IF
END_ACTION

ACTION visit:
//////////////////////////////////////////////////
//perform single visit motion					//
//////////////////////////////////////////////////

IF initStateLVL2 = FALSE THEN
	initStateLVL2 := TRUE;
	stateLVL2 :=2010;
	motionBusy := TRUE;
END_IF	

CASE stateLVL2 OF

	2010: 
		motionBusy := TRUE;
		GVL.fbWaitTimer(IN:=TRUE, PT:=GVL.expoTime,);
		axis[XM].mcMoveAbs(Axis:=axis[XM].axisRef, Position:= POS_END_C, Velocity:=speed, Execute:=TRUE);
		IF GVL.fbWaitTimer.Q THEN
			axis[XP].mcMoveAbs(Axis:=axis[XP].axisRef, Position:= POS_END_C, Velocity:=speed, Execute:=TRUE);
		END_IF
		IF axis[XP].mcMoveAbs.Done AND axis[XM].mcMoveAbs.Done THEN
			GVL.fbWaitTimer(IN:=FALSE);
			axis[XP].mcMoveAbs(Axis:=axis[XP].axisRef, Execute:=FALSE);
			axis[XM].mcMoveAbs(Axis:=axis[XM].axisRef, Execute:=FALSE);
			stateLVL2:=2020;
		END_IF
		
	2020:
		GVL.fbWaitTimer(IN:=TRUE, PT:=T#500MS,);
		IF GVL.fbWaitTimer.Q THEN
			GVL.fbWaitTimer(IN:=FALSE);
			stateLVL2:=2030;
		END_IF
		
	2030: 
		GVL.fbWaitTimer(IN:=TRUE, PT:=GVL.expoTime,);
		axis[XP].mcMoveAbs(Axis:=axis[XP].axisRef, Position:= POS_START_C, Velocity:=speed, Execute:=TRUE);
		IF GVL.fbWaitTimer.Q THEN
			axis[XM].mcMoveAbs(Axis:=axis[XM].axisRef, Position:= POS_START_C, Velocity:=speed, Execute:=TRUE);
		END_IF
		IF axis[XP].mcMoveAbs.Done AND axis[XM].mcMoveAbs.Done THEN
			GVL.fbWaitTimer(IN:=FALSE);
			axis[XP].mcMoveAbs(Axis:=axis[XP].axisRef, Execute:=FALSE);
			axis[XM].mcMoveAbs(Axis:=axis[XM].axisRef, Execute:=FALSE);
			stateLVL2:=2040;
		END_IF	

		
	2040: //End action
		initStateLVL2 := FALSE;
		stateLVL2 := 0;
		motionBusy := FALSE;
END_CASE
END_ACTION

END_FUNCTION_BLOCK

(* stored: Version 1.1.0.1, ProductVersion 3.1.4020.12
   POU TestMotion: Id {f5ec753e-2f53-4143-ab85-291d0817da2d}, SpecialFunc None
   Action calibrateXM: Id {f55b06c7-6108-4c5a-8395-ce4a40ab5ee7}
   Action calibrateXP: Id {79108831-3b18-418a-a130-e890c3b4b0b4}
   Action closeShutterMinus: Id {c8eebc4c-d2a0-42de-82dc-8e5673de86c8}
   Action closeShutterPlus: Id {43ef5e05-4492-480d-abe4-6a35baea3693}
   Action cycler: Id {b3bb7fae-23b4-40ef-bb63-00745722aa1f}
   Action homeShutter: Id {68ff6a15-67b8-44ff-b25f-ff9ce5a24dba}
   Action openShutter: Id {f7febd62-8f52-4abd-992a-fedae8687624}
   Action tracking: Id {f70340f7-7c55-4a6a-973e-20bf0bb509c6}
   Action visit: Id {afd9cbcc-4d11-4009-8c14-8d9062a035ea} *)
